TYPE ST_HMI_Monitor_Powerstack :
STRUCT
	// stack
	r_Powerload					: REAL;
	r_DcPower					: REAL;
	r_ActivePower				: REAL;
	r_throttlingValue			: REAL;
	
	b_ACDetected				: BOOL;
	b_DCDetected				: BOOL;
	b_StartedState				: BOOL;
	b_islandOperation			: BOOL;
	b_ControlEnabled			: BOOL;
	e_NetContState				: eNetContactorState;
	e_ACrotationState			: eACRotationState;
	e_StatusPowerStack			: eStatusPowerstack;
	
	//Master
	b_MasterEnabled				: BOOL;
	b_MasterWarning				: BOOL;
	b_MasterMCCBfb				: BOOL;
	e_MasterState				: eStatusPowerModule;
	r_MasterthrotValue			: REAL;
	b_MasterTempThrotActive		: BOOL;
	b_MasterCurrThrotActive		: BOOL;		
	
	
	b_SlaveEnabled				: BOOL;
	b_SlaveWarning				: BOOL;
	b_SlaveMCCBfb				: BOOL;
	e_SlaveState				: eStatusPowerModule;
	r_SlavethrotValue			: REAL;
	b_SlaveTempThrotActive		: BOOL;
	b_SlaveCurrThrotActive		: BOOL;		
	
END_STRUCT
END_TYPE

(* stored: Version 1.1.0.1, ProductVersion 3.1.4026.18
   DUT ST_HMI_Monitor_Powerstack: Id {088b3e40-0f06-41c3-813c-ec133fa95505} *)
